FUNCTION ArrayContains : BOOL;
VAR_INPUT
	arr : POINTER TO BYTE;
	arrSize : UDINT;
	element : POINTER TO BYTE;
	typeSize : UDINT;
END_VAR
VAR_OUTPUT
	index : UDINT;
END_VAR
VAR
	i : UDINT;
END_VAR

FOR i:=0 TO arrSize-1 BY typeSize DO
	
	IF MEMCMP(arr[i], element, typeSize) = 0 THEN
		index := i;
		ArrayContains := TRUE;
		RETURN;
	END_IF
	
END_FOR

END_FUNCTION

(* stored: Version 1.1.0.1, ProductVersion 3.1.4024.11
   POU ArrayContains: Id {81112d19-78a8-48e5-969a-18eef3df6033}, SpecialFunc None *)
